{attribute 'GeneratedUsingTerminal: EL2521-0124-0018'}
{attribute addProperty BoxType "EL2521-0124-0018"}
{attribute addProperty Id "Enable_PLSBOOL1OutputBOOL1"}
{attribute addProperty CRC "2005331871"}
{attribute addProperty Size "2"}
TYPE Control_7786EF9F :
STRUCT
	{attribute addProperty Name "Enable_PLS"}
	Enable_PLS : BOOL;
	{attribute addProperty Name "Output"}
	Output : BOOL;
END_STRUCT
END_TYPE

(* stored: Version 1.2.0.0, ProductVersion 3.1.4024.9
   DUT Control_7786EF9F: Id {8eba1bac-646b-4c37-a830-9968452e4454} *)
